TYPE SlotHeader :
STRUCT
END_STRUCT
END_TYPE

(* stored: Version 1.1.0.1, ProductVersion 3.1.4020.12
   DUT SlotHeader: Id {e698adb5-cbc9-437a-b2b6-14deb728af6c} *)
